TYPE "TrkMng_Row"
VERSION : 0.1
// Block: TrkMng_Row
   STRUCT
      Visible : Bool;
      RowColor : Int;
      PNum : Int;
      IDPiece : UDInt;
      PartProgram : DInt;
      Sum_Result : Trk_AreaResult;
   END_STRUCT;

END_TYPE
